Staubli VAL3: isDetected.pgx

public program isDetected(num& x_nHowMany[])
begin
  x_nHowMany=nNumOfPart
end
